// TIA Portal V17 export
// export: Created 2025-03-10T12:15:08.4333453Z, ExportSetting WithDefaults, DisplayName Totally Integrated Automation Portal, DisplayVersion V17 Update 8, DisplayName TIA Portal Openness, DisplayVersion V17 Update 8, DisplayName TIA Portal Version Control Interface, DisplayVersion V17, DisplayName SINAMICS Startdrive Advanced, DisplayVersion V17 SP2, DisplayName SINAMICS Startdrive G110M, G120, G120C, G120D, G120P, G115D, DisplayVersion V17 SP2, DisplayName SINAMICS Startdrive G130, G150, S120, S150, SINAMICS MV, S210, DisplayVersion V17 SP2, DisplayName STEP 7 Professional, DisplayVersion V17 Update 8, DisplayName SINUMERIK ONE STEP 7 Toolbox, DisplayVersion V17 Update 12, DisplayName SINUMERIK 840D sl STEP 7 Toolbox, DisplayVersion V17 Update 12, DisplayName STEP 7 Safety, DisplayVersion V17 Update 6, DisplayName WinCC Advanced, DisplayVersion V17 Update 8
FUNCTION "FC8006_UNIT_02_PART_STATUS_FULL_DEPTH" : Void   // FC8006, LAD
{ S7_Optimized_Access := 'TRUE' }
VERSION : 0.1
// stored: AutoNumber false, IsIECCheckEnabled false, SetENOAutomatically false, UDAEnableTagReadback false
BEGIN

REGION Network 1: FIXTURE 1 PART STATUS UNIT 02
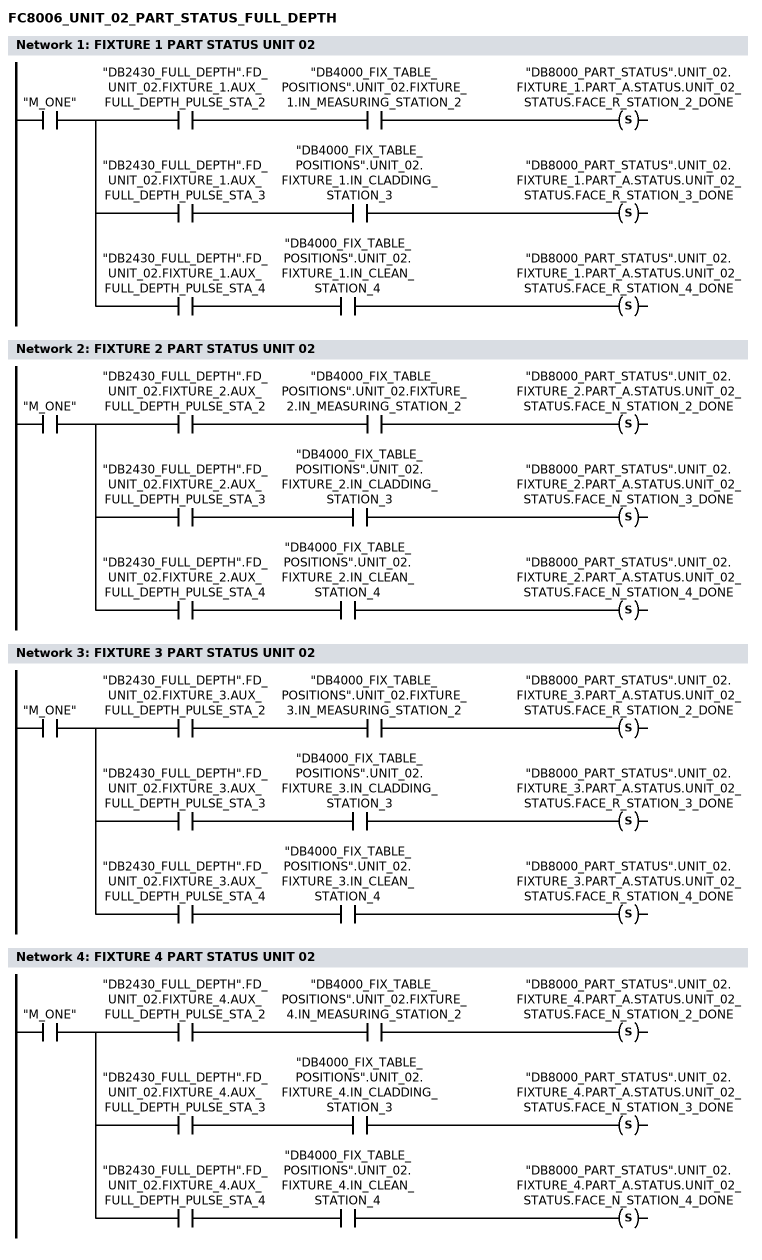
   RUNG wire#powerrail
      Contact( "M_ONE" )
      wire#w1
      Contact( "DB2430_FULL_DEPTH".FD_UNIT_02.FIXTURE_1.AUX_FULL_DEPTH_PULSE_STA_2 )
      Contact( "DB4000_FIX_TABLE_POSITIONS".UNIT_02.FIXTURE_1.IN_MEASURING_STATION_2 )
      S_Coil( "DB8000_PART_STATUS".UNIT_02.FIXTURE_1.PART_A.STATUS.UNIT_02_STATUS.FACE_R_STATION_2_DONE )
   END_RUNG
   RUNG wire#w1
      Contact( "DB2430_FULL_DEPTH".FD_UNIT_02.FIXTURE_1.AUX_FULL_DEPTH_PULSE_STA_3 )
      Contact( "DB4000_FIX_TABLE_POSITIONS".UNIT_02.FIXTURE_1.IN_CLADDING_STATION_3 )
      S_Coil( "DB8000_PART_STATUS".UNIT_02.FIXTURE_1.PART_A.STATUS.UNIT_02_STATUS.FACE_R_STATION_3_DONE )
   END_RUNG
   RUNG wire#w1
      Contact( "DB2430_FULL_DEPTH".FD_UNIT_02.FIXTURE_1.AUX_FULL_DEPTH_PULSE_STA_4 )
      Contact( "DB4000_FIX_TABLE_POSITIONS".UNIT_02.FIXTURE_1.IN_CLEAN_STATION_4 )
      S_Coil( "DB8000_PART_STATUS".UNIT_02.FIXTURE_1.PART_A.STATUS.UNIT_02_STATUS.FACE_R_STATION_4_DONE )
   END_RUNG
   // the same network as SCL:
   IF "M_ONE" AND "DB2430_FULL_DEPTH".FD_UNIT_02.FIXTURE_1.AUX_FULL_DEPTH_PULSE_STA_2 AND "DB4000_FIX_TABLE_POSITIONS".UNIT_02.FIXTURE_1.IN_MEASURING_STATION_2 THEN
       "DB8000_PART_STATUS".UNIT_02.FIXTURE_1.PART_A.STATUS.UNIT_02_STATUS.FACE_R_STATION_2_DONE := TRUE;
   END_IF;
   IF "M_ONE" AND "DB2430_FULL_DEPTH".FD_UNIT_02.FIXTURE_1.AUX_FULL_DEPTH_PULSE_STA_3 AND "DB4000_FIX_TABLE_POSITIONS".UNIT_02.FIXTURE_1.IN_CLADDING_STATION_3 THEN
       "DB8000_PART_STATUS".UNIT_02.FIXTURE_1.PART_A.STATUS.UNIT_02_STATUS.FACE_R_STATION_3_DONE := TRUE;
   END_IF;
   IF "M_ONE" AND "DB2430_FULL_DEPTH".FD_UNIT_02.FIXTURE_1.AUX_FULL_DEPTH_PULSE_STA_4 AND "DB4000_FIX_TABLE_POSITIONS".UNIT_02.FIXTURE_1.IN_CLEAN_STATION_4 THEN
       "DB8000_PART_STATUS".UNIT_02.FIXTURE_1.PART_A.STATUS.UNIT_02_STATUS.FACE_R_STATION_4_DONE := TRUE;
   END_IF;
END_REGION

REGION Network 2: FIXTURE 2 PART STATUS UNIT 02
   RUNG wire#powerrail
      Contact( "M_ONE" )
      wire#w1
      Contact( "DB2430_FULL_DEPTH".FD_UNIT_02.FIXTURE_2.AUX_FULL_DEPTH_PULSE_STA_2 )
      Contact( "DB4000_FIX_TABLE_POSITIONS".UNIT_02.FIXTURE_2.IN_MEASURING_STATION_2 )
      S_Coil( "DB8000_PART_STATUS".UNIT_02.FIXTURE_2.PART_A.STATUS.UNIT_02_STATUS.FACE_N_STATION_2_DONE )
   END_RUNG
   RUNG wire#w1
      Contact( "DB2430_FULL_DEPTH".FD_UNIT_02.FIXTURE_2.AUX_FULL_DEPTH_PULSE_STA_3 )
      Contact( "DB4000_FIX_TABLE_POSITIONS".UNIT_02.FIXTURE_2.IN_CLADDING_STATION_3 )
      S_Coil( "DB8000_PART_STATUS".UNIT_02.FIXTURE_2.PART_A.STATUS.UNIT_02_STATUS.FACE_N_STATION_3_DONE )
   END_RUNG
   RUNG wire#w1
      Contact( "DB2430_FULL_DEPTH".FD_UNIT_02.FIXTURE_2.AUX_FULL_DEPTH_PULSE_STA_4 )
      Contact( "DB4000_FIX_TABLE_POSITIONS".UNIT_02.FIXTURE_2.IN_CLEAN_STATION_4 )
      S_Coil( "DB8000_PART_STATUS".UNIT_02.FIXTURE_2.PART_A.STATUS.UNIT_02_STATUS.FACE_N_STATION_4_DONE )
   END_RUNG
   // the same network as SCL:
   IF "M_ONE" AND "DB2430_FULL_DEPTH".FD_UNIT_02.FIXTURE_2.AUX_FULL_DEPTH_PULSE_STA_2 AND "DB4000_FIX_TABLE_POSITIONS".UNIT_02.FIXTURE_2.IN_MEASURING_STATION_2 THEN
       "DB8000_PART_STATUS".UNIT_02.FIXTURE_2.PART_A.STATUS.UNIT_02_STATUS.FACE_N_STATION_2_DONE := TRUE;
   END_IF;
   IF "M_ONE" AND "DB2430_FULL_DEPTH".FD_UNIT_02.FIXTURE_2.AUX_FULL_DEPTH_PULSE_STA_3 AND "DB4000_FIX_TABLE_POSITIONS".UNIT_02.FIXTURE_2.IN_CLADDING_STATION_3 THEN
       "DB8000_PART_STATUS".UNIT_02.FIXTURE_2.PART_A.STATUS.UNIT_02_STATUS.FACE_N_STATION_3_DONE := TRUE;
   END_IF;
   IF "M_ONE" AND "DB2430_FULL_DEPTH".FD_UNIT_02.FIXTURE_2.AUX_FULL_DEPTH_PULSE_STA_4 AND "DB4000_FIX_TABLE_POSITIONS".UNIT_02.FIXTURE_2.IN_CLEAN_STATION_4 THEN
       "DB8000_PART_STATUS".UNIT_02.FIXTURE_2.PART_A.STATUS.UNIT_02_STATUS.FACE_N_STATION_4_DONE := TRUE;
   END_IF;
END_REGION

REGION Network 3: FIXTURE 3 PART STATUS UNIT 02
   RUNG wire#powerrail
      Contact( "M_ONE" )
      wire#w1
      Contact( "DB2430_FULL_DEPTH".FD_UNIT_02.FIXTURE_3.AUX_FULL_DEPTH_PULSE_STA_2 )
      Contact( "DB4000_FIX_TABLE_POSITIONS".UNIT_02.FIXTURE_3.IN_MEASURING_STATION_2 )
      S_Coil( "DB8000_PART_STATUS".UNIT_02.FIXTURE_3.PART_A.STATUS.UNIT_02_STATUS.FACE_R_STATION_2_DONE )
   END_RUNG
   RUNG wire#w1
      Contact( "DB2430_FULL_DEPTH".FD_UNIT_02.FIXTURE_3.AUX_FULL_DEPTH_PULSE_STA_3 )
      Contact( "DB4000_FIX_TABLE_POSITIONS".UNIT_02.FIXTURE_3.IN_CLADDING_STATION_3 )
      S_Coil( "DB8000_PART_STATUS".UNIT_02.FIXTURE_3.PART_A.STATUS.UNIT_02_STATUS.FACE_R_STATION_3_DONE )
   END_RUNG
   RUNG wire#w1
      Contact( "DB2430_FULL_DEPTH".FD_UNIT_02.FIXTURE_3.AUX_FULL_DEPTH_PULSE_STA_4 )
      Contact( "DB4000_FIX_TABLE_POSITIONS".UNIT_02.FIXTURE_3.IN_CLEAN_STATION_4 )
      S_Coil( "DB8000_PART_STATUS".UNIT_02.FIXTURE_3.PART_A.STATUS.UNIT_02_STATUS.FACE_R_STATION_4_DONE )
   END_RUNG
   // the same network as SCL:
   IF "M_ONE" AND "DB2430_FULL_DEPTH".FD_UNIT_02.FIXTURE_3.AUX_FULL_DEPTH_PULSE_STA_2 AND "DB4000_FIX_TABLE_POSITIONS".UNIT_02.FIXTURE_3.IN_MEASURING_STATION_2 THEN
       "DB8000_PART_STATUS".UNIT_02.FIXTURE_3.PART_A.STATUS.UNIT_02_STATUS.FACE_R_STATION_2_DONE := TRUE;
   END_IF;
   IF "M_ONE" AND "DB2430_FULL_DEPTH".FD_UNIT_02.FIXTURE_3.AUX_FULL_DEPTH_PULSE_STA_3 AND "DB4000_FIX_TABLE_POSITIONS".UNIT_02.FIXTURE_3.IN_CLADDING_STATION_3 THEN
       "DB8000_PART_STATUS".UNIT_02.FIXTURE_3.PART_A.STATUS.UNIT_02_STATUS.FACE_R_STATION_3_DONE := TRUE;
   END_IF;
   IF "M_ONE" AND "DB2430_FULL_DEPTH".FD_UNIT_02.FIXTURE_3.AUX_FULL_DEPTH_PULSE_STA_4 AND "DB4000_FIX_TABLE_POSITIONS".UNIT_02.FIXTURE_3.IN_CLEAN_STATION_4 THEN
       "DB8000_PART_STATUS".UNIT_02.FIXTURE_3.PART_A.STATUS.UNIT_02_STATUS.FACE_R_STATION_4_DONE := TRUE;
   END_IF;
END_REGION

REGION Network 4: FIXTURE 4 PART STATUS UNIT 02
   RUNG wire#powerrail
      Contact( "M_ONE" )
      wire#w1
      Contact( "DB2430_FULL_DEPTH".FD_UNIT_02.FIXTURE_4.AUX_FULL_DEPTH_PULSE_STA_2 )
      Contact( "DB4000_FIX_TABLE_POSITIONS".UNIT_02.FIXTURE_4.IN_MEASURING_STATION_2 )
      S_Coil( "DB8000_PART_STATUS".UNIT_02.FIXTURE_4.PART_A.STATUS.UNIT_02_STATUS.FACE_N_STATION_2_DONE )
   END_RUNG
   RUNG wire#w1
      Contact( "DB2430_FULL_DEPTH".FD_UNIT_02.FIXTURE_4.AUX_FULL_DEPTH_PULSE_STA_3 )
      Contact( "DB4000_FIX_TABLE_POSITIONS".UNIT_02.FIXTURE_4.IN_CLADDING_STATION_3 )
      S_Coil( "DB8000_PART_STATUS".UNIT_02.FIXTURE_4.PART_A.STATUS.UNIT_02_STATUS.FACE_N_STATION_3_DONE )
   END_RUNG
   RUNG wire#w1
      Contact( "DB2430_FULL_DEPTH".FD_UNIT_02.FIXTURE_4.AUX_FULL_DEPTH_PULSE_STA_4 )
      Contact( "DB4000_FIX_TABLE_POSITIONS".UNIT_02.FIXTURE_4.IN_CLEAN_STATION_4 )
      S_Coil( "DB8000_PART_STATUS".UNIT_02.FIXTURE_4.PART_A.STATUS.UNIT_02_STATUS.FACE_N_STATION_4_DONE )
   END_RUNG
   // the same network as SCL:
   IF "M_ONE" AND "DB2430_FULL_DEPTH".FD_UNIT_02.FIXTURE_4.AUX_FULL_DEPTH_PULSE_STA_2 AND "DB4000_FIX_TABLE_POSITIONS".UNIT_02.FIXTURE_4.IN_MEASURING_STATION_2 THEN
       "DB8000_PART_STATUS".UNIT_02.FIXTURE_4.PART_A.STATUS.UNIT_02_STATUS.FACE_N_STATION_2_DONE := TRUE;
   END_IF;
   IF "M_ONE" AND "DB2430_FULL_DEPTH".FD_UNIT_02.FIXTURE_4.AUX_FULL_DEPTH_PULSE_STA_3 AND "DB4000_FIX_TABLE_POSITIONS".UNIT_02.FIXTURE_4.IN_CLADDING_STATION_3 THEN
       "DB8000_PART_STATUS".UNIT_02.FIXTURE_4.PART_A.STATUS.UNIT_02_STATUS.FACE_N_STATION_3_DONE := TRUE;
   END_IF;
   IF "M_ONE" AND "DB2430_FULL_DEPTH".FD_UNIT_02.FIXTURE_4.AUX_FULL_DEPTH_PULSE_STA_4 AND "DB4000_FIX_TABLE_POSITIONS".UNIT_02.FIXTURE_4.IN_CLEAN_STATION_4 THEN
       "DB8000_PART_STATUS".UNIT_02.FIXTURE_4.PART_A.STATUS.UNIT_02_STATUS.FACE_N_STATION_4_DONE := TRUE;
   END_IF;
END_REGION
END_FUNCTION
